PROGRAM P_Demo_F_BA_GetDateTime
VAR
    fnReturn                       : ST_BA_DateTime; // 返回值
END_VAR

// =============================================================================
// Tc3_BA2_Common.F_BA_GetDateTime 演示程序
// =============================================================================
// 场景：快速获取"当前时刻"作为时间戳；用于报警 / 趋势记录。
//
// 价值：一行 FC 替代调用 `FB_LocalSystemTime` 等异步 FB 的复杂用法。
//
// 验证：登录 PLC 后，按例程内变量在线写值；监视输出 / 返回值，结合 §1 功能
//       简述的预期行为对照（详见配套 .md 文档 §7 业务场景）。
//
// 验证步骤：
//   1. 右键 PLC 项目下 POUs 文件夹 → Add → Existing Item → 选本 .TcPOU 文件
//   2. 引用 Tc3_BA2_Common（References → Add library）
//   3. 编译 → 登录 → 运行；按上方『验证』指引在线写值观察
// =============================================================================

fnReturn := F_BA_GetDateTime();

END_PROGRAM

(* stored: Version 1.1.0.1, ProductVersion 3.1.4024.5
   POU P_Demo_F_BA_GetDateTime: Id {e03e75f1-6908-5f3c-a1b3-349065912689}, SpecialFunc None *)
